// TIA Portal V20 export
FUNCTION_BLOCK "FB_Digita_Inputs"   // FB1, LAD
{ S7_Optimized_Access := 'TRUE' }
// stored: MemoryReserve 100, SetENOAutomatically false
   VAR_INPUT
      "I-Digital_Input_0" : Bool;
      "I-Digital_Input_1" : Bool;
      "I-Digital_Input_2" : Bool;
      "I-Digital_Input_3" : Bool;
      "I-Digital_Input_4" : Bool;
      "I-Digital_Input_5" : Bool;
      "I-Digital_Input_6" : Bool;
      "I-Digital_Input_7" : Bool;
      "I-Digital_Input_8" : Bool;
      "I-Digital_Input_9" : Bool;
      "I-Digital_Input_10" : Bool;
      "I-Digital_Input_11" : Bool;
      "I-Digital_Input_12" : Bool;
      "I-Digital_Input_13" : Bool;
   END_VAR
   VAR_OUTPUT
      DB_Digital_Input_0 : Bool;
      DB_Digital_Input_1 : Bool;
      DB_Digital_Input_2 : Bool;
      DB_Digital_Input_3 : Bool;
      DB_Digital_Input_4 : Bool;
      DB_Digital_Input_5 : Bool;
      DB_Digital_Input_6 : Bool;
      DB_Digital_Input_7 : Bool;
      DB_Digital_Input_8 : Bool;
      DB_Digital_Input_9 : Bool;
      DB_Digital_Input_10 : Bool;
      DB_Digital_Input_11 : Bool;
      DB_Digital_Input_12 : Bool;
      DB_Digital_Input_13 : Bool;
   END_VAR
BEGIN

REGION Network 1
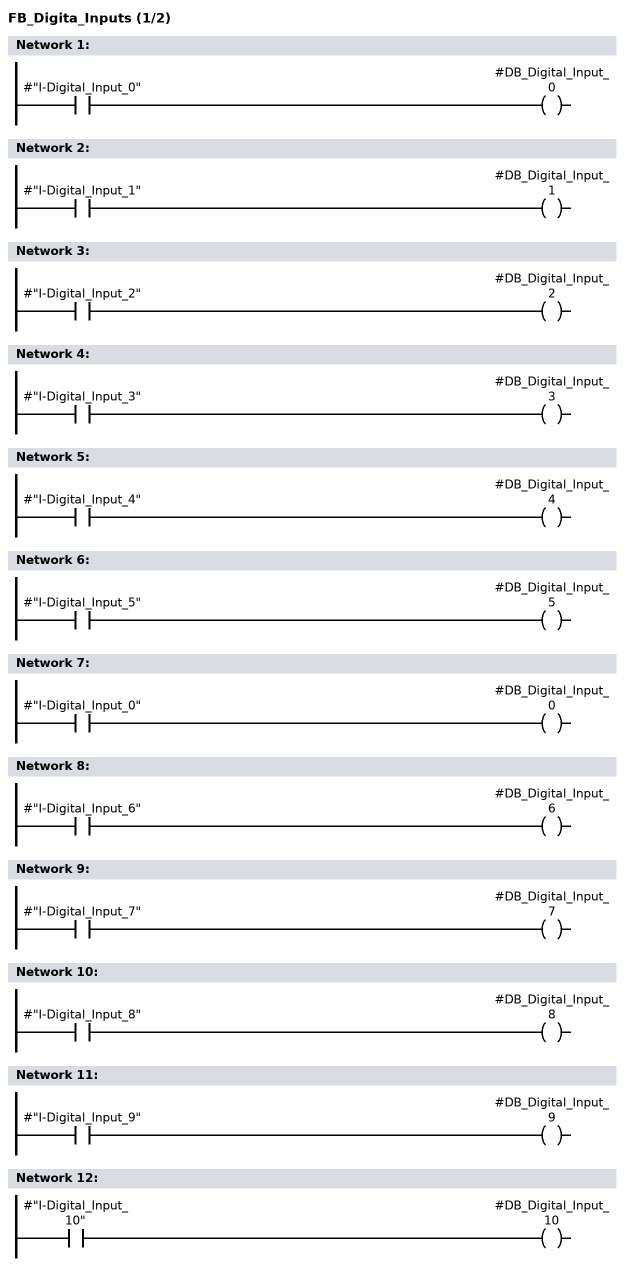
   RUNG wire#powerrail
      Contact( #"I-Digital_Input_0" )
      Coil( #DB_Digital_Input_0 )
   END_RUNG
   // the same network as SCL:
   #DB_Digital_Input_0 := #"I-Digital_Input_0";
END_REGION

REGION Network 2
   RUNG wire#powerrail
      Contact( #"I-Digital_Input_1" )
      Coil( #DB_Digital_Input_1 )
   END_RUNG
   // the same network as SCL:
   #DB_Digital_Input_1 := #"I-Digital_Input_1";
END_REGION

REGION Network 3
   RUNG wire#powerrail
      Contact( #"I-Digital_Input_2" )
      Coil( #DB_Digital_Input_2 )
   END_RUNG
   // the same network as SCL:
   #DB_Digital_Input_2 := #"I-Digital_Input_2";
END_REGION

REGION Network 4
   RUNG wire#powerrail
      Contact( #"I-Digital_Input_3" )
      Coil( #DB_Digital_Input_3 )
   END_RUNG
   // the same network as SCL:
   #DB_Digital_Input_3 := #"I-Digital_Input_3";
END_REGION

REGION Network 5
   RUNG wire#powerrail
      Contact( #"I-Digital_Input_4" )
      Coil( #DB_Digital_Input_4 )
   END_RUNG
   // the same network as SCL:
   #DB_Digital_Input_4 := #"I-Digital_Input_4";
END_REGION

REGION Network 6
   RUNG wire#powerrail
      Contact( #"I-Digital_Input_5" )
      Coil( #DB_Digital_Input_5 )
   END_RUNG
   // the same network as SCL:
   #DB_Digital_Input_5 := #"I-Digital_Input_5";
END_REGION

REGION Network 7
   RUNG wire#powerrail
      Contact( #"I-Digital_Input_0" )
      Coil( #DB_Digital_Input_0 )
   END_RUNG
   // the same network as SCL:
   #DB_Digital_Input_0 := #"I-Digital_Input_0";
END_REGION

REGION Network 8
   RUNG wire#powerrail
      Contact( #"I-Digital_Input_6" )
      Coil( #DB_Digital_Input_6 )
   END_RUNG
   // the same network as SCL:
   #DB_Digital_Input_6 := #"I-Digital_Input_6";
END_REGION

REGION Network 9
   RUNG wire#powerrail
      Contact( #"I-Digital_Input_7" )
      Coil( #DB_Digital_Input_7 )
   END_RUNG
   // the same network as SCL:
   #DB_Digital_Input_7 := #"I-Digital_Input_7";
END_REGION

REGION Network 10
   RUNG wire#powerrail
      Contact( #"I-Digital_Input_8" )
      Coil( #DB_Digital_Input_8 )
   END_RUNG
   // the same network as SCL:
   #DB_Digital_Input_8 := #"I-Digital_Input_8";
END_REGION

REGION Network 11
   RUNG wire#powerrail
      Contact( #"I-Digital_Input_9" )
      Coil( #DB_Digital_Input_9 )
   END_RUNG
   // the same network as SCL:
   #DB_Digital_Input_9 := #"I-Digital_Input_9";
END_REGION

REGION Network 12
   RUNG wire#powerrail
      Contact( #"I-Digital_Input_10" )
      Coil( #DB_Digital_Input_10 )
   END_RUNG
   // the same network as SCL:
   #DB_Digital_Input_10 := #"I-Digital_Input_10";
END_REGION

REGION Network 13
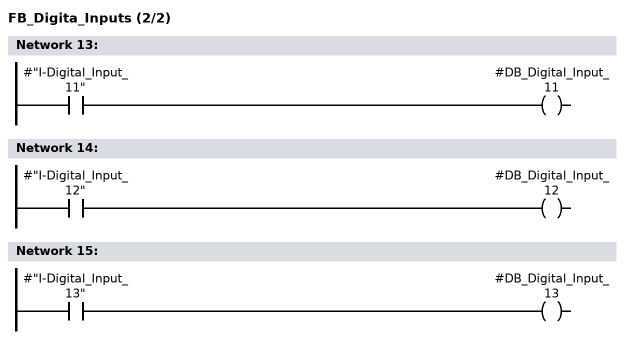
   RUNG wire#powerrail
      Contact( #"I-Digital_Input_11" )
      Coil( #DB_Digital_Input_11 )
   END_RUNG
   // the same network as SCL:
   #DB_Digital_Input_11 := #"I-Digital_Input_11";
END_REGION

REGION Network 14
   RUNG wire#powerrail
      Contact( #"I-Digital_Input_12" )
      Coil( #DB_Digital_Input_12 )
   END_RUNG
   // the same network as SCL:
   #DB_Digital_Input_12 := #"I-Digital_Input_12";
END_REGION

REGION Network 15
   RUNG wire#powerrail
      Contact( #"I-Digital_Input_13" )
      Coil( #DB_Digital_Input_13 )
   END_RUNG
   // the same network as SCL:
   #DB_Digital_Input_13 := #"I-Digital_Input_13";
END_REGION
END_FUNCTION_BLOCK
